(* IEC 61131-3 sources: POMIRTS_lab3/AS/Library/AsPPP, 3 files *)

(* ---- AsPPP.typ ---- *)
(********************************************************************
 * COPYRIGHT -- Bernecker + Rainer
 ********************************************************************
 * Library: AsPPP
 * File: AsPPP.typ
 * Author: B+R
 ********************************************************************
 * Data types of library AsPPP
 ********************************************************************)

TYPE
    pppPARAMETER_typ	: STRUCT		(*ppp parameter*)
		pHostAddr		: UDINT;		(*pointer to the host ip address (string format)*)
		pPeerAddr		: UDINT;		(*pointer to the peer ip address (string format)*)
		pOptions		: UDINT;		(*pointer to the ppp otions struct (optional)*)
		pSecrets		: UDINT;		(*pointer to the secret table (optional)*)
		sectablen		: UDINT;		(*number of entries in the secrets table*)
	END_STRUCT;
END_TYPE

(* ---- AsPPP.fun ---- *)
(********************************************************************
 * COPYRIGHT -- Bernecker + Rainer
 ********************************************************************
 * Library: AsPPP
 * File: AsPPP.fun
 * Author: B+R
 ********************************************************************
 * Functions and function blocks of library AsPPP
 ********************************************************************)

FUNCTION_BLOCK PPPStart					(*starts a ppp device; asynchronous execution*)
	VAR_INPUT
		enable			: BOOL;			(*enables execution*)
		pDevice			: UDINT;		(*device name given as a pointer, e.g., "SL<x>.SS<y>.IF<z>"*)
		pDeviceParam	: UDINT;		(*pointer to the parent device parameter (optional)*)
		pPppParam		: UDINT;		(*pointer to the ppp parameter*)
	END_VAR
	VAR
        i_state			: UINT;			(*internal variable*)
		i_result		: UINT;			(*internal variable*)
        i_tmp			: UDINT;		(*internal variable*)
	END_VAR
	VAR_OUTPUT
		status			: UINT;			(*execution status: ERR_OK, ERR_FUB_ENABLE_FALSE, ERR_FUB_BUSY, 0xXXXX = see help*)
	END_VAR
END_FUNCTION_BLOCK

FUNCTION_BLOCK PPPStop					(*stops a ppp device; asynchronous execution*)
	VAR_INPUT
		enable			: BOOL;			(*enables execution*)
		pDevice			: UDINT;		(*device name given as a pointer, e.g., "SL<x>.SS<y>.IF<z>"*)
	END_VAR

	VAR
        i_state			: UINT;			(*internal variable*)
		i_result		: UINT;			(*internal variable*)
        i_tmp			: UDINT;		(*internal variable*)
	END_VAR

	VAR_OUTPUT
		status			: UINT;			(*execution status: ERR_OK, ERR_FUB_ENABLE_FALSE, ERR_FUB_BUSY, 0xXXXX = see help*)
	END_VAR
END_FUNCTION_BLOCK

(* ---- AsPPP.var ---- *)
(********************************************************************
 * COPYRIGHT -- Bernecker + Rainer
 ********************************************************************
 * Library: AsPPP
 * File: AsPPP.var
 * Author: B+R
 ********************************************************************
 * Local variables of library AsPPP
 ********************************************************************)

VAR CONSTANT
	pppERR_INVALID_DEVICE				: UINT := 32000;	(*invlalid parent device*)
END_VAR
